Fanuc KAREL source: kt00747.KL

-- PROVISIONAL review KL for V770-1; original PC SHA256 0baa17bd99441a2a2b366ae2ca747710b8e7b9fa5e8a29acf541ac6a43b0e43b
-- Incomplete behavior may be omitted. Consult companion uncertainty JSON. Do not deploy.
PROGRAM KT00747
%NOLOCKGROUP
BEGIN
  -- UNRESOLVED_PC offsets 5-18; opcodes 22,1D,23
  -- UNRESOLVED_PC offsets 23-27; opcodes 7F
END KT00747
